{attribute 'qualified_only'}
{attribute 'strict'}
TYPE E_MotorDOL :
(
	enum_member := 0
);
END_TYPE

(* stored: Version 1.1.0.1, ProductVersion 3.1.4024.12
   DUT E_MotorDOL: Id {0660cc86-54ba-44ee-9954-a90f6ebf4cbb} *)
